// TIA Portal V19 export
FUNCTION_BLOCK "Projekt2B_RobotGrinder"   // FB1, STL
{ S7_Optimized_Access := 'TRUE' }
// stored: MemoryReserve 100
   VAR_INPUT
      Emergency_Stop_Status_150K1 : Bool;
      Sensor_102B2 : Bool;
      Sensor_102B3 : Bool;
      Sensor_102B4 : Bool;
      Sensor_102B5 : Bool;
      Sensor_102B6 : Bool;
      Reset : Bool;
   END_VAR
   VAR_OUTPUT
      Valve_106Q6 : Bool;
      Motor_4Q3 : Bool;
      Motor_4Q5 : Bool;
      Motor_6Q1 : Bool;
      Motor_6Q3 : Bool;
      Reset_Safety_150K1 : Bool;
   END_VAR
BEGIN
END_FUNCTION_BLOCK
